// TIA Portal V20 export
DATA_BLOCK "ET200SP_204"   // DB296
// stored: MemoryReserve 100
   VAR
      "SP204.00 Main OP: Emergency stop" : Bool;
      SPARE1 : Bool;
      SPARE2 : Bool;
      SPARE3 : Bool;
      RESERVED : Bool;
      SPARE4 : Bool;
      SPARE5 : Bool;
      SPARE6 : Bool;
   END_VAR
BEGIN
END_DATA_BLOCK
